% RSLogix 500 project TEST_BAK005.RSS, saved by version 11.00.00.00 %
PROJECT "UNTITLED"    % processor: MicroLogix 1000 %

PROGRAM FILES
  LAD 2 "MAIN_PROG"  4 rungs
  LAD 3 "USER_FAULT"  1 rungs
  LAD 4 "HSC_INT"  1 rungs
  LAD 5 "STI_INT"  1 rungs
  LAD 6, 7, 8, 9, 10, 11, 12, 13, 14, 15, 16: only END

DATA FILES
  O0 OUTPUT  1 elements
  I1 INPUT  2 elements
  S2 STATUS  33 elements
  B3 BINARY  32 elements
  T4 TIMER  40 elements
  C5 COUNTER  32 elements
  R6 CONTROL  16 elements
  N7 INTEGER  105 elements

LADDER 2 "MAIN_PROG"
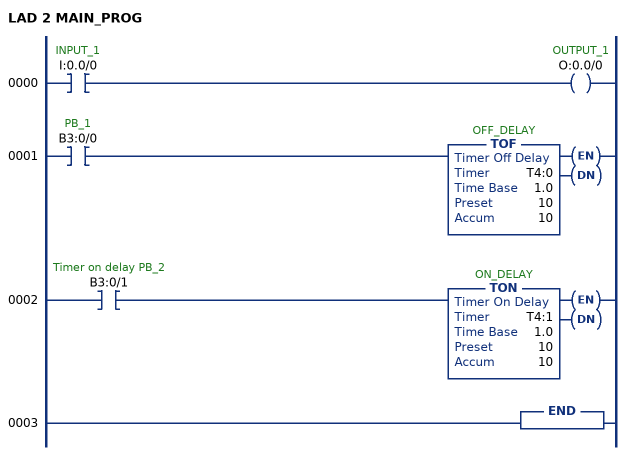
% Rung: 0 %
SOR XIC I:0.0/0 OTE O:0.0/0 EOR
%   I:0.0/0  INPUT_1 %
%   O:0.0/0  OUTPUT_1 %
% Rung: 1 %
SOR XIC B3:0/0 TOF T4:0 1.0 10 10 EOR
%   B3:0/0  PB_1 %
%   T4:0  OFF_DELAY %
% Rung: 2 %
SOR XIC B3:0/1 TON T4:1 1.0 10 10 EOR
%   B3:0/1  PB_2  "Timer on delay" %
%   T4:1  ON_DELAY %
% Rung: 3 %
SOR END EOR

DATA TABLE (non-zero values as saved)
DATA B3
% B3:0 % 0X0002 0X0000 0X0000 0X0000 0X0000 0X0000 0X0000 0X0000 0X0000 0X0000
DATA T4
% .PRE .ACC %
% T4:0 % 10 10
% T4:1 % 10 10
